# EPICS substitutions: BLDApp/Db/IOC-SYS0-BD02bsa.substitutions
#==============================================================================
#
# Abs:  LCLS Beam Synchronous Acquisition records for SYS0 BD02
#
# Name: IOC-SYS0-BD02bsa.substitutions
#
# Associated Displays: bsa_sys0_maint.edl
#
# Rem:  Instantiate one line for every beam synchronous item.
#
# Macros:
#	DEVICE	Name of the beam synchronous triggered device.  Must match the
#		name in <ioc>trig.substitutions without the 3rd colon and beyond.
#	LOC	IOC location.
#	UN	IOC unit number.
#	IOC	Name of IOC that contains the EVR, not including the 3rd colon.
#	ATRB    BSA attribute name
#	IN	Input to BSA record
#	SLCLNK	Set to "" if the IOC is not slc-aware.
#		Otherwise, set to "<device>:FANOUTSLC".
#==============================================================================
#
file bsaBLDEdef.db {
    pattern
    { DEVICE, LOC, UN, SLCLNK, BPM1, BPM2}
    { BLD:SYS0:600, SYS0, 600, "", LTU_235, LTU_370 }
}
